FUNCTION_BLOCK FB_BarnDoors
VAR_INPUT
    bladeA  : UINT;
    bladeB  : UINT;
    gap     : UINT;
    fClosedGap  : LREAL;
    fBladeSize  : LREAL;
    
END_VAR
VAR_OUTPUT
END_VAR
VAR
    iState: INT;
    fPositionToSet : LREAL;
    fCalculatedPosition : REAL;
    fCalculatedInt AT %Q* : DINT;
    fbCalcGap : FB_CalculateGap;
    fbCalcAngle : FB_CalculateAngle;
    
    timeout: TON;
END_VAR

timeout.PT:=T#2S; //2second timeout to attempt rehomes
timeout();
//Geometry check
(*Position values outside the allowable range defined by the blade geometry cannot be reached but will result in errors during calculation*)
//Check upper limit
IF GVL.astAxes[gap].stConfig.fPosition > (2*fBladeSize+fClosedGap) THEN
    GVL.astAxes[gap].stConfig.fPosition:= 2*fBladeSize+fClosedGap;
END_IF
//Check lower limit
IF GVL.astAxes[gap].stConfig.fPosition < (fClosedGap) THEN
    GVL.astAxes[gap].stConfig.fPosition:= fClosedGap;
END_IF

//Check switches and enables (wouldn't cause crash)
IF GVL.astAxes[bladeA].stStatus.bBwEnabled AND GVL.astAxes[bladeB].stStatus.bFwEnabled THEN
    GVL.astAxes[gap].stInputs.bLimitFwd:= TRUE;
ELSE
    GVL.astAxes[gap].stInputs.bLimitFwd:= FALSE;
END_IF

IF GVL.astAxes[bladeA].stStatus.bFwEnabled AND GVL.astAxes[bladeB].stStatus.bBwEnabled THEN
    GVL.astAxes[gap].stInputs.bLimitBwd:= TRUE;
ELSE
    GVL.astAxes[gap].stInputs.bLimitBwd:= FALSE;
END_IF

IF GVL.astAxes[bladeA].stStatus.bEnabled AND GVL.astAxes[bladeB].stStatus.bEnabled THEN
    GVL.astAxes[gap].stControl.bEnable:= TRUE;
ELSE
    GVL.astAxes[gap].stControl.bEnable:= FALSE;
END_IF

fbCalcAngle(GapSize:=GVL.astAxes[gap].stConfig.fPosition);

CASE iState OF
0://Wait for blade axes enabled
    IF GVL.astAxes[bladeA].stStatus.bEnabled AND GVL.astAxes[bladeB].stStatus.bEnabled THEN
        iState:=1;
	END_IF

1:
    IF (NOT GVL.astAxes[bladeA].stStatus.bHomed) OR (NOT GVL.astAxes[bladeB].stStatus.bHomed) THEN
        GVL.astAxes[bladeA].stControl.eCommand:=E_MotionFunctions.eHome;
        GVL.astAxes[bladeA].stControl.bExecute:=TRUE;
        GVL.astAxes[bladeB].stControl.eCommand:=E_MotionFunctions.eHome;
        GVL.astAxes[bladeB].stControl.bExecute:=TRUE;
	END_IF
    iState:= 2;

2://Wait for all axes calibrated, if bladeA AND bladeB calibrated, can direct home gap to the correct value
    IF (GVL.astAxes[bladeA].stStatus.bHomed AND GVL.astAxes[bladeB].stStatus.bHomed) THEN
        fbCalcGap(AngleBladeA:=GVL.astAxes[bladeA].stStatus.fActPosition,AngleBladeB:=GVL.astAxes[bladeB].stStatus.fActPosition,fBladeSize:= fBladeSize, fClosedGap:=fClosedGap);
        GVL.astAxes[gap].stControl.eCommand:= E_MotionFunctions.eHome;
        GVL.astAxes[gap].stConfig.eHomeSeq:= E_HomingRoutines.eHomeDirect;
        GVL.astAxes[gap].stConfig.fHomePosition:= fbCalcGap.GapSize;
        GVL.astAxes[gap].stControl.bExecute:=TRUE;
        iState:=3;
        timeout.IN:=TRUE;
    END_IF
    
3://Wait for calibration complete
    //IF (GVL.astAxes[bladeA].stStatus.bHomed) AND (GVL.astAxes[bladeB].stStatus.bHomed) THEN
        //iState:=10;    
    IF (GVL.astAxes[gap].stStatus.bHomed) THEN
        iState:=10;
	END_IF
    IF timeout.Q THEN
        timeout.IN:=FALSE;
        iState:=0;
	END_IF
    
10://Everything calibrated, start intercepting absolute position moves
//Check for absolute position move of virtual axis and issue move to blades if move executed
IF GVL.astAxes[gap].stControl.eCommand = E_MotionFunctions.eMoveAbsolute AND GVL.astAxes[gap].stControl.bExecute AND GVL.astAxes[gap].stStatus.bEnabled THEN
    fbCalcAngle(GapSize:=GVL.astAxes[gap].stConfig.fPosition);
    GVL.astAxes[bladeA].stControl.eCommand := E_MotionFunctions.eMoveAbsolute;
    GVL.astAxes[bladeA].stConfig.fPosition := fbCalcAngle.AngleBladeB;
    GVL.astAxes[bladeA].stConfig.fVelocity:=GVL.astAxes[gap].stConfig.fVelocity;
    GVL.astAxes[bladeA].stControl.bExecute:=TRUE;
    GVL.astAxes[bladeB].stControl.eCommand := E_MotionFunctions.eMoveAbsolute;
    GVL.astAxes[bladeB].stConfig.fPosition := fbCalcAngle.AngleBladeA;
    GVL.astAxes[bladeB].stConfig.fVelocity:=GVL.astAxes[gap].stConfig.fVelocity;
    GVL.astAxes[bladeB].stControl.bExecute:=TRUE;
END_IF


999: //ERROR STATE
    GVL.astAxes[gap].stControl.bEnable:= FALSE;
    //Wait for reset of axes and block moves.
    IF NOT(GVL.astAxes[bladeA].stStatus.bError AND GVL.astAxes[bladeB].stStatus.bError) THEN
        iState:=0;
	END_IF
    
END_CASE

IF GVL.astAxes[bladeA].stStatus.bError OR GVL.astAxes[bladeB].stStatus.bError THEN
    iState:=999;
END_IF

END_FUNCTION_BLOCK

(* stored: Version 1.1.0.1, ProductVersion 3.1.4024.0
   POU FB_BarnDoors: Id {b6c2e4cf-4c7d-4459-a188-0564af6adf0d}, SpecialFunc None *)
